FUNCTION_BLOCK SW_FormatWstring
//格式化字符串
//SwenChen
//20171123
VAR_INPUT
	WstringIn:			WSTRING;
	D1:					DINT;
	D2:					DINT;
	S1:					STRING;
END_VAR
VAR_OUTPUT
	WstringOUT:			WSTRING;
END_VAR
VAR
	Var1: 				INT;
END_VAR


Var1:=WFIND(WstringIn,"%D");
IF Var1<>0 THEN
	WstringOUT := WREPLACE(WstringIn,DINT_TO_WSTRING(D1),2,Var1);

	Var1:=WFIND(WstringOUT,"%D");
	IF Var1<>0 THEN
		WstringOUT := WREPLACE(WstringOUT,DINT_TO_WSTRING(D2),2,Var1);
	END_IF
ELSE
	WstringOUT:=WstringIN;
END_IF

Var1:=WFIND(WstringOUT,"%S");
IF Var1<>0 THEN
	WstringOUT := WREPLACE(WstringOUT,STRING_TO_WSTRING(S1),2,Var1);
END_IF

END_FUNCTION_BLOCK

(* stored: Version 1.1.0.1, ProductVersion 3.1.4024.12
   POU SW_FormatWstring: Id {26730b47-e2ce-4ffe-9d4b-72ef26749fd2}, SpecialFunc None *)
